FUNCTION_BLOCK RandomUniform IMPLEMENTS IRandom
VAR
  _lowerBound : LREAL;
  _upperBound : LREAL;  
  _rnd : Tc2_System.DRAND;
END_VAR

METHOD FB_init : BOOL
VAR_INPUT
	bInitRetains : BOOL; // if TRUE, the retain variables are initialized (warm start / cold start)
	bInCopyCode : BOOL;  // if TRUE, the instance afterwards gets moved into the copy code (online change)
  seed : INT;      
  lowerBound : LREAL;
  upperBound : LREAL;
END_VAR
SetSeed(seed);
SetBounds(lowerBound, upperBound);
END_METHOD

METHOD Next : LREAL
_rnd();
Next := _rnd.Num * (_upperBound-_lowerBound) + _lowerBound;
END_METHOD

METHOD FINAL SetBounds
VAR_INPUT
  lowerBound : LREAL;
  upperBound : LREAL;
END_VAR
_lowerBound := lowerBound;
_upperBound := upperBound;
END_METHOD

METHOD FINAL SetSeed
VAR_INPUT
  seed : INT;
END_VAR
_rnd.Seed := seed;
END_METHOD

END_FUNCTION_BLOCK

(* stored: Version 1.1.0.1
   POU RandomUniform: Id {fa774a23-5e02-49ec-9016-716b5ff60699}, SpecialFunc None
   Method FB_init: Id {9a9c39d2-635b-448a-bc73-f477997a62a2}
   Method Next: Id {fc1d4962-bd25-43e6-8b66-8b256f2ef9e4}
   Method SetBounds: Id {205ca8e8-8f72-4eda-a540-2e345c889383}
   Method SetSeed: Id {14683bec-6f11-44ca-94c8-c6276f35f8ea} *)
